{attribute 'GeneratedUsingTerminal: EL3773-0000-0017'}
{attribute addProperty BoxType "EL3773-0000-0017"}
{attribute addProperty Id "I1_STATUSAT %I*I1_STATUS_B07533568"}
{attribute addProperty CRC "2313189400"}
{attribute addProperty Size "8"}
TYPE L1_Current_Status_89E07818 :
STRUCT
	{attribute addProperty Name "I1_STATUS"}
	I1_STATUS AT %I* : I1_STATUS_B0753356;
END_STRUCT
END_TYPE

(* stored: Version 1.2.0.0, ProductVersion 3.1.4024.9
   DUT L1_Current_Status_89E07818: Id {01edfd5d-19c2-4d9c-9880-1492049a4421} *)
